FUNCTION NextStep : UDINT
VAR_IN_OUT
	StateVar : UDINT;
END_VAR

NextStep := StateVar := ((StateVar / 10) * 10) + 10;

END_FUNCTION

(* stored: Version 1.1.0.1
   POU NextStep: Id {655f2740-2d13-0edf-3108-02757fda7453}, SpecialFunc None *)
